TYPE TestSlaveConfigData :
STRUCT
	config1 : INT;
	config2 : INT;
END_STRUCT
END_TYPE

(* stored: Version 1.1.0.1, ProductVersion 3.1.4024.12
   DUT TestSlaveConfigData: Id {cdc02899-ce84-4fa4-8056-f91342d074e8} *)
